Omron CX-Programmer project NewProject (CX-Programmer 9.73)

# PLC NewPLC1: CP2E-N N

## Global symbols (name address type ; comment)
0 CHANNEL  ; MOTOR1
0.00 BOOL  ; LAMP 1
0.01 BOOL  ; BUTTON 1
0.02 BOOL  ; BUTTON2
0.03 BOOL  ; BUTTON3
100.00 BOOL  ; LAMP2
100.01 BOOL  ; DIR Motor1
100.02 BOOL  ; DIR1
100.03 BOOL  ; LAMP3
100.04 BOOL  ; BREAK1
100.05 BOOL  ; BREAK2
100.06 BOOL  ; EN1
D0 CHANNEL  ; MOTOR1
D40 CHANNEL  ; INI M1
D50 CHANNEL  ; SAVE SET POINT
W0.00 BOOL  ; B_1
W0.01 BOOL  ; B_2
W0.02 BOOL  ; B_2
W0.03 BOOL  ; CW M1
W0.04 BOOL  ; CCW M1
W0.05 BOOL  ; BUTTON_SAVE

## Program NewProgram1 (cyclic task 0)
Local symbols
HOME_M1 D80 UINT  ; Home Motor 1
HOME_M2 D81 UINT  ; Home Motor 2
POSITION D83 UINT  ; CORDINAT POSITION
SET_POINT D82 UINT  ; SET POINT TEACHING

### Section Set_Motor

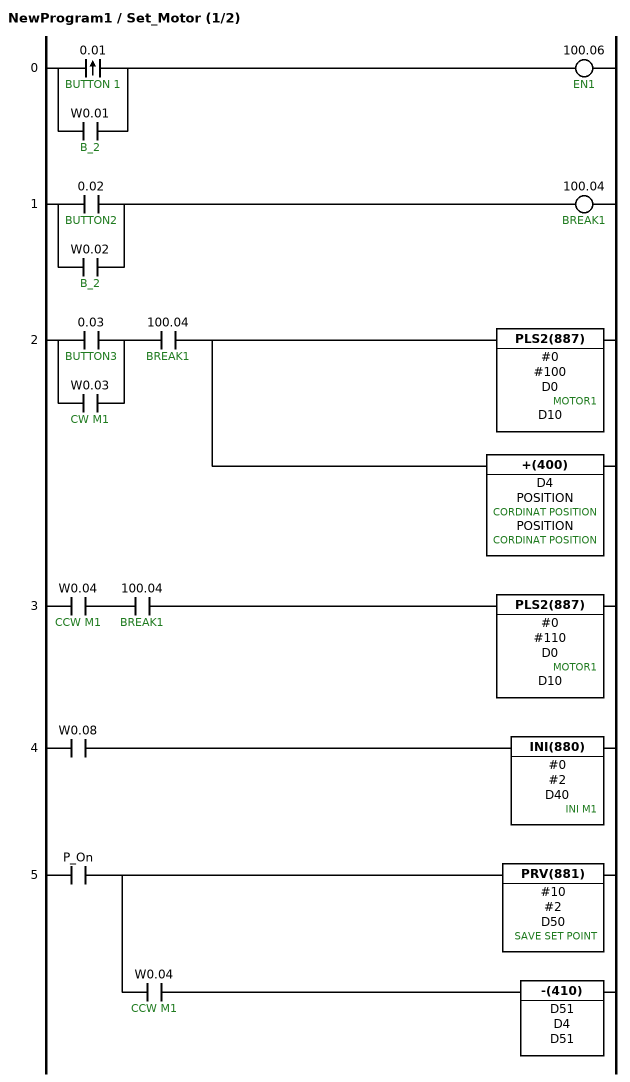
; rung 0
@LD 0.01  ; BUTTON 1
OR W0.01  ; B_2
OUT 100.06  ; EN1
; rung 1
LD 0.02  ; BUTTON2
OR W0.02  ; B_2
OUT 100.04  ; BREAK1
; rung 2
LD 0.03  ; BUTTON3
OR W0.03  ; CW M1
AND 100.04  ; BREAK1
PLS2(887) #0 #100 D0 D10  ; MOTOR1
+(400) D4 POSITION POSITION  ; CORDINAT POSITION
; rung 3
LD W0.04  ; CCW M1
AND 100.04  ; BREAK1
PLS2(887) #0 #110 D0 D10  ; MOTOR1
; rung 4
LD W0.08
INI(880) #0 #2 D40  ; INI M1
; rung 5
LD P_On
PRV(881) #10 #2 D50  ; SAVE SET POINT
AND W0.04  ; CCW M1
-(410) D51 D4 D51

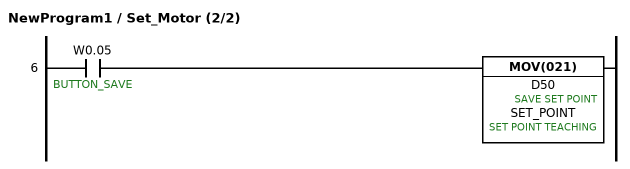
; rung 6
LD W0.05  ; BUTTON_SAVE
MOV(021) D50 SET_POINT  ; SAVE SET POINT, SET POINT TEACHING

### Section Section2

### Section Section3
; rung 0
END(001)